ABB RobotStudio station: Project.rspag

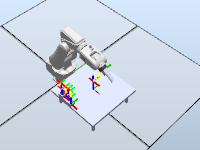
--- station ---
Station RA_2022_ABB_PROJEKAT (saved by RobotStudio 7.0.8732.594)
Controller IRB120_3_58
  mechanical unit ROB_1: IRB120_3_58__01, 6 joints, base frame (0, 0, 0) mm
Layout (positions relative to the parent item):
  - IRB120_3_58__01 [mechanism, from Robots\IRB120_3_58_G_01.rslib] at (0, 0, 0) mm; joint values [0, 0.4511, -0.3041, 0, 0.3766, 0] (rad or m)
  - Sto [part] at (630, -250, 0) mm
  - DrzacPapira [part] at (337.16, -241.74, 175) mm, rotated rx 90 ry 0 rz 180 deg
  - OdlaganjePapira [part] at (318.58, -233.58, 175) mm, rotated rx 90 ry 0 rz 0 deg
  - Alat [part] at (489.06, 0, 522) mm, rotated rx 180 ry 60 rz 180 deg
Attachment: Alat is attached to IRB120_3_58__01 / Link6

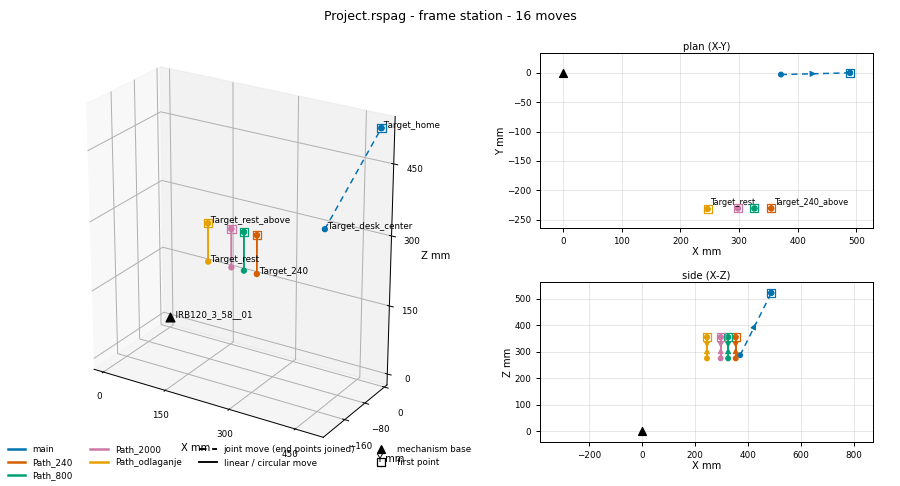
[picture p0: tool path of Project.rspag in frame station, 16 of 21 moves have a stored position in this frame; points joined in program order, loops and branches not executed]
--- Backups/IRB120_3_58/RAPID/TASK1/PROGMOD/CalibData.mod ---
MODULE CalibData
	PERS wobjdata Centar_stola:=[FALSE,TRUE,"",[[371.428,-2.973,175],[1,0,0,0]],[[0,0,112],[1,0,0,0]]];
	PERS wobjdata Odlaganje:=[FALSE,TRUE,"",[[266.015,-243.107,225],[1,0,0,0]],[[0,0,0],[1,0,0,0]]];
	PERS wobjdata Preuzimanje:=[FALSE,TRUE,"",[[366.377,-246.724,205],[1,0,0,0]],[[0,0,0],[1,0,0,0]]];
ENDMODULE

--- Backups/IRB120_3_58/RAPID/TASK1/PROGMOD/Module1.mod ---
MODULE Module1
    CONST robtarget Target_home:=[[489.061487217,0,522],[0.5,0,0.866025404,0],[0,0,0,0],[9E+09,9E+09,9E+09,9E+09,9E+09,9E+09]];
    CONST robtarget Target_240_above:=[[-11.563209766,15.710086064,150],[0,0,1,0],[0,0,0,0],[9E+09,9E+09,9E+09,9E+09,9E+09,9E+09]];
    CONST robtarget Target_240:=[[-11.563209766,15.710086064,70],[0,0,1,0],[0,0,0,0],[9E+09,9E+09,9E+09,9E+09,9E+09,9E+09]];
    CONST robtarget Target_800_above:=[[-40.199209766,15.710086064,150],[0,0,1,0],[0,0,0,0],[9E+09,9E+09,9E+09,9E+09,9E+09,9E+09]];
    CONST robtarget Target_800:=[[-40.199209766,15.710086064,70],[0,0,1,0],[0,0,0,0],[9E+09,9E+09,9E+09,9E+09,9E+09,9E+09]];
    CONST robtarget Target_2000_above:=[[-68.274209766,15.710086064,150],[0,0,1,0],[0,0,0,0],[9E+09,9E+09,9E+09,9E+09,9E+09,9E+09]];
    CONST robtarget Target_2000:=[[-68.274209766,15.710086064,70],[0,0,1,0],[0,0,0,0],[9E+09,9E+09,9E+09,9E+09,9E+09,9E+09]];
    CONST robtarget Target_rest_above:=[[-19.626016678,11.004870974,130],[0,0,1,0],[-1,0,-1,0],[9E+09,9E+09,9E+09,9E+09,9E+09,9E+09]];
    CONST robtarget Target_rest:=[[-19.626016678,11.004870974,50],[0,0,1,0],[-1,0,-1,0],[9E+09,9E+09,9E+09,9E+09,9E+09,9E+09]];
    CONST robtarget Target_desk_center:=[[0,0,0],[0,0,1,0],[0,0,0,0],[9E+09,9E+09,9E+09,9E+09,9E+09,9E+09]];
!***********************************************************
    !
    ! Module:  Module1
    !
    ! Description:
    !   Predmet: Robotika i automatizacija
    !   Projekat 1
    !
    ! Authors: Vukotic Djuro, Krunic Aleksa
    !
    ! Version: 1.0
    !
    !***********************************************************


LOCAL FUNC num Random()
    VAR num nSeed:=320;
    VAR num nSeed_age:=150;
    CONST num nModulus:=655;
    CONST num nMultiplier:=251;
    CONST num nIncrement:=13849;
    IF nSeed_age>140 THEN
        nSeed:=GetTime(\Sec)*GetTime(\Min);
        nSeed_age:=0;
    ENDIF
    nSeed_age:=nSeed_age+1;
    nSeed:=((nMultiplier*Abs(nSeed))+nIncrement) MOD nModulus;
    RETURN (nSeed/nModulus);
ENDFUNC

PROC cameraFunction( VAR num objShape, VAR num firstDim, VAR num secondDim, VAR num objOrient)
    VAR num tmp;
    tmp:=Random();

    IF tmp <= 0.33 THEN
        objShape:= 0;
        tmp:=Random();
        firstDim:= 150 + tmp*150;
        secondDim:= 150 + tmp*150;
        tmp:=Random();
        objOrient:= -180 + tmp*280;
    ELSEIF tmp >=0.66 THEN
        objShape:=1;
        tmp:=Random();
        firstDim:= 150 + tmp*150;
        WaitTime 1;
        tmp:=Random();
        secondDim:= 150 + tmp*150;
        WaitTime 1;
        tmp:=Random();
        objOrient:= -180 + tmp*280;
    ELSE
        objShape:=2;
        tmp:=Random();
        firstDim:= 150 + tmp*150;
        secondDim:= 150 + tmp*150;
        objOrient:= 0;
    ENDIF
ENDPROC

! Main programa
    PROC main()
        !Pravljenje promenljivih koje korisnik treba da unese i inicijalizacija digitalnog izlaza
        VAR num Paper_granulation;
        VAR num Overlap_percentage;
        VAR num objShape;
        VAR num firstDim;
        VAR num secondDim;
        VAR num objOrient;
        VAR robtarget Target_temp;
        VAR num Remaining_width;
        VAR num Sign;

        WHILE 1>0 DO
        ! Resetovanje digitalnih izlaza
        SetDO AttachPaper, 0;
        SetDO P240, 0;
        SetDO P800, 0;
        SetDO P2000, 0;

        ! Unos granulacije papira i procenta preklapanja
        TPErase;
        IspravkaG: TPReadNum Paper_granulation, "Uneti granulaciju papira. Za prekid programa uneti -1";
        IF Paper_granulation = -1 THEN
            TPWrite "Program ce se ugasiti za 5 sekundi";
            WaitTime 5;
            Break;
        ENDIF
        IF Paper_granulation <> 240 AND Paper_granulation <> 800 AND Paper_granulation <> 2000 THEN
            TPWrite "Nepostojeca granulacija. Izabrati izmedju granulacija 240, 800 i 2000";
            GOTO IspravkaG;
        ENDIF
        TPWrite " ";
        IspravkaP: TPReadNum Overlap_percentage, "Uneti procenat preklapanja";
        IF Overlap_percentage <> 0 AND Overlap_percentage <> 25 AND Overlap_percentage <> 50 THEN
            TPWrite "Procenat preklapanja moze biti 0%, 25% ili 50%";
            GOTO IspravkaP;
        ENDIF
        TPWrite " ";

        ! Postupak uzimanja papira i informisanje korisnika o papiru koji se koristi za proces smirglanja
        IF Paper_granulation = 240 THEN
            Path_240;
            TPWrite "Papir granulacije 240 se koristi";
        ELSEIF Paper_granulation = 800 THEN
            Path_800;
            TPWrite "Papir granulacije 800 se koristi";
        ELSEIF Paper_granulation = 2000 THEN
            Path_2000;
            TPWrite "Papir granulacije 2000 se koristi";
        ENDIF
        TPWrite " ";

        ! Simulacija kamere koja detektuje oblik i dimenzije ploce
        cameraFunction objShape,firstDim,secondDim, objOrient;

        ! Ispisivanje dimenzija i orijentacije ploce
        IF objShape = 0 THEN
            TPWrite "Oblik: KVADRAT ";
        ELSEIF objShape = 1 THEN
            TPWrite "Oblik: PRAVOUGAONIK ";
        ELSE
            TPWrite "Oblik: KRUG ";
        ENDIF
        !TPWrite "Oblik ", \Num:=objShape;
        TPWrite "Prva dimenzija ", \Num:=firstDim;
        TPWrite "Druga dimenzija ", \Num:=secondDim;
        TPWrite "Orijentacija "\Num:=objOrient;
        TPWrite " ";

        ! Dozvola za pocetak smirglanja
        ! TPWrite "Ceka se dozvola za pocetak smirglanja.  Pritisnite dugme -";
        ! WaitDI StartProces,1;

        ! Proces smirglanja
        Target_temp:=Target_desk_center;
        MoveJ Target_home,v1000,z100,tool0\WObj:=wobj0;
        MoveJ Target_temp,v1000,z0,tool0\WObj:=Centar_stola;
        firstDim:=firstDim-28;
        secondDim:=secondDim-28;
        MoveJ RelTool (Target_temp, 0, 0, 0 \Rz:= -objOrient),v100,fine,tool0\WObj:=Centar_stola;
        Target_temp :=  RelTool (Target_temp, 0, 0, 0 \Rz:= -objOrient);
        MoveJ Offs(Target_temp, Cos(-objOrient)*(-firstDim/2)-Sin(-objOrient)*(-secondDim/2),Sin(-objOrient)*(-firstDim/2)+Cos(-objOrient)*(-secondDim/2),0),v100,fine,tool0\WObj:=Centar_stola;
        Target_temp:=Offs(Target_temp, Cos(-objOrient)*(-firstDim/2)-Sin(-objOrient)*(-secondDim/2),Sin(-objOrient)*(-firstDim/2)+Cos(-objOrient)*(-secondDim/2),0);
        Remaining_width:=secondDim;
        Sign:=1;
        WHILE Remaining_width>0 DO
            MoveL Offs(Target_temp, Cos(-objOrient)*(Sign*firstDim)-Sin(-objOrient)*(0),Sin(-objOrient)*(Sign*firstDim)+Cos(-objOrient)*(0), 0),v100,fine,tool0\WObj:=Centar_stola;
            Target_temp:=Offs(Target_temp, Cos(-objOrient)*(Sign*firstDim)-Sin(-objOrient)*(0),Sin(-objOrient)*(Sign*firstDim)+Cos(-objOrient)*(0), 0);
            MoveL Offs(Target_temp, Cos(-objOrient)*(0)-Sin(-objOrient)*((28-Overlap_percentage/100*28)),Sin(-objOrient)*(0)+Cos(-objOrient)*((28-Overlap_percentage/100*28)), 0),v100,fine,tool0\WObj:=Centar_stola;
            Target_temp:=Offs(Target_temp, Cos(-objOrient)*(0)-Sin(-objOrient)*((28-Overlap_percentage/100*28)),Sin(-objOrient)*(0)+Cos(-objOrient)*((28-Overlap_percentage/100*28)), 0);
            Remaining_width:=Remaining_width-28+Overlap_percentage/100*28;
            Sign:=Sign*(-1);
        ENDWHILE
        MoveJ Target_desk_center,v100,z0,tool0\WObj:=Centar_stola;
        MoveJ Target_home,v1000,z100,tool0\WObj:=wobj0;

        ! Odlaganje
        Path_odlaganje;
        MoveJ Target_home,v1000,z100,tool0\WObj:=wobj0;
        ENDWHILE

    ENDPROC
    PROC Path_240()
        MoveJ Target_240_above,v1000,z0,tool0\WObj:=Preuzimanje;
        MoveL Target_240,v100,fine,tool0\WObj:=Preuzimanje;
        SetDO AttachPaper, 1;
        WaitTime \InPos, 1;
        SetDO P240, 1;
        MoveL Target_240_above,v100,fine,tool0\WObj:=Preuzimanje;
    ENDPROC
    PROC Path_800()
        MoveJ Target_800_above,v1000,z0,tool0\WObj:=Preuzimanje;
        MoveL Target_800,v100,fine,tool0\WObj:=Preuzimanje;
        SetDO AttachPaper, 1;
        WaitTime \InPos, 1;
        SetDO P800, 1;
        MoveL Target_800_above,v100,fine,tool0\WObj:=Preuzimanje;
    ENDPROC
    PROC Path_2000()
        MoveJ Target_2000_above,v1000,z0,tool0\WObj:=Preuzimanje;
        MoveL Target_2000,v100,fine,tool0\WObj:=Preuzimanje;
        SetDO AttachPaper, 1;
        WaitTime \InPos, 1;
        SetDO P2000, 1;
        MoveL Target_2000_above,v100,fine,tool0\WObj:=Preuzimanje;
    ENDPROC
    PROC Path_odlaganje()
        MoveJ Target_rest_above,v1000,z10,tool0\WObj:=Odlaganje;
        MoveL Target_rest,v100,z10,tool0\WObj:=Odlaganje;
        SetDO AttachPaper, 0;
        MoveL Target_rest_above,v100,z10,tool0\WObj:=Odlaganje;
    ENDPROC
ENDMODULE

--- Backups/IRB120_3_58/RAPID/TASK1/PROGMOD/RsTempModule.mod ---
MODULE RsTempModule
PROC RsTempPath()
ENDPROC

ENDMODULE

--- Backups/IRB120_3_58/SYSPAR/EIO.cfg ---
EIO:CFG_1.0:6:1::
#
EIO_SIGNAL:

      -Name "P240" -SignalType "DO"

      -Name "P800" -SignalType "DO"

      -Name "P2000" -SignalType "DO"

      -Name "AttachPaper" -SignalType "DO"

      -Name "StartProces" -SignalType "DI"
